(* CODESYS project backup.export

Project tree, tasks and I/O mapping:
  Device : CODESYS Control Win V3 x64, CODESYS, version 3.5.21.10
    application Application
      libraries: Standard, 3.5.18.0 (System)
      task MainTask (cyclic, interval t#20ms, priority 1) calls PLC_PRG
      data type E_Command
      data type E_States
      global variables GVL
      global variables GV_IO
      function BitsToByte [ST]
      function block FB_CircularQueue_Command [ST]: Clear, Dequeue, Enqueue, Peek
      function block FB_ConveyorController [ST]
      function block FB_MachineCenter [ST]: bBusy, bDoorOpened, bEnable, bError, bProduceLids, Progress
      function block FB_OperatorPanel [?]
      function block FB_Positioner [ST]: Clamp, Lift, Lower, Release
      function block FB_PusherController [ST]: Execute
      function block FB_RunTimeTracker [ST]
      function block FB_TwoAxisPaP [ST]: IsMoving, MoveXNeg, MoveXPos, PickUp, ProcessCommand, PutDown
      function block FB_VisionSensorAD [ST]
      program PLC_PRG [ST]
      function block Stage1_PartDetection [ST]: ProcessObjectDetection
      function block Stage2_MC [ST]: ReadyForPart
      function block Stage3_Assembly [ST]
      Symbols
      global variables PersistentVars
    Ethernet : Ethernet, CODESYS, version 4.2.0.0
        settings: IPAddress = [127,0,0,1]; SubnetMask = [255,255,255,0]; GatewayAddress = [0,0,0,0]; MACAddress = [16#00,16#00,16#00,16#00,16#00,16#00]; SaveCommunicationSettings = FALSE; IPAddress = [192,168,0,2]; SubnetMask = [255,255,255,0]; GatewayAddress = [0,0,0,0]
      ModbusTCP_Server_Device : ModbusTCP Server Device, CODESYS, version 4.4.0.0
          settings: DistinctBitAreas = TRUE; Coils Size = 24; Discrete Inputs Size = 19
          input  Application.GV_IO.iMC_Progress : WORD  // Holding Registers.Holding Registers
          input  Application.GV_IO.iBaseVisionSensorBit0 : BOOL  // Coils.Coils.Bit0
          input  Application.GV_IO.iBaseVisionSensorBit1 : BOOL  // Coils.Coils.Bit1
          input  Application.GV_IO.iBaseVisionSensorBit2 : BOOL  // Coils.Coils.Bit2
          input  Application.GV_IO.iBaseVisionSensorBit3 : BOOL  // Coils.Coils.Bit3
          input  Application.GV_IO.iBasePusherBackLimit : BOOL  // Coils.Coils.Bit4
          input  Application.GV_IO.iBasePusherFrontLimit : BOOL  // Coils.Coils.Bit5
          input  Application.GV_IO.iBaseDiffuseSensor : BOOL  // Coils.Coils.Bit6
          input  Application.GV_IO.iEmergencyStopButton : BOOL  // Coils.Coils.Bit7
          input  Application.GV_IO.iResetButton : BOOL  // Coils.Coils.Bit0
          input  Application.GV_IO.iStartButton : BOOL  // Coils.Coils.Bit1
          input  Application.GV_IO.iStopButton : BOOL  // Coils.Coils.Bit2
          input  Application.GV_IO.iMC_Busy : BOOL  // Coils.Coils.Bit3
          input  Application.GV_IO.iMC_Error : BOOL  // Coils.Coils.Bit4
          input  Application.GV_IO.iLidAtPositioner : BOOL  // Coils.Coils.Bit5
          input  Application.GV_IO.iMC_Opened : BOOL  // Coils.Coils.Bit6
          input  Application.GV_IO.iBaseAtPositioner : BOOL  // Coils.Coils.Bit7
          input  Application.GV_IO.iContainerAtExit : BOOL  // Coils.Coils.Bit0
          input  Application.GV_IO.iBasePositionerLimit : BOOL  // Coils.Coils.Bit1
          input  Application.GV_IO.iLidPositionerLimit : BOOL  // Coils.Coils.Bit2
          input  Application.GV_IO.iPaPPartDetected : BOOL  // Coils.Coils.Bit3
          input  Application.GV_IO.iPaPMovingX : BOOL  // Coils.Coils.Bit4
          input  Application.GV_IO.iPaPMovingZ : BOOL  // Coils.Coils.Bit5
          input  Application.GV_IO.iBasePositionerClamped : BOOL  // Coils.Coils.Bit6
          input  Application.GV_IO.iLidPositionerClamped : BOOL  // Coils.Coils.Bit7
          output Application.GV_IO.oResetButtonLight : BOOL  // Discrete Inputs.Discrete Inputs.Bit0
          output Application.GV_IO.oBasePusher : BOOL  // Discrete Inputs.Discrete Inputs.Bit1
          output Application.GV_IO.oStageOneConveyor : BOOL  // Discrete Inputs.Discrete Inputs.Bit2
          output Application.GV_IO.oStartButtonLight : BOOL  // Discrete Inputs.Discrete Inputs.Bit3
          output Application.GV_IO.oStopButtonLight : BOOL  // Discrete Inputs.Discrete Inputs.Bit4
          output Application.GV_IO.oProcessOnLight : BOOL  // Discrete Inputs.Discrete Inputs.Bit5
          output Application.GV_IO.oMC_Start : BOOL  // Discrete Inputs.Discrete Inputs.Bit6
          output Application.GV_IO.oMC_Stop : BOOL  // Discrete Inputs.Discrete Inputs.Bit7
          output Application.GV_IO.oMC_Reset : BOOL  // Discrete Inputs.Discrete Inputs.Bit0
          output Application.GV_IO.oMC_ProduceLids : BOOL  // Discrete Inputs.Discrete Inputs.Bit1
          output Application.GV_IO.oBaseConveyor : BOOL  // Discrete Inputs.Discrete Inputs.Bit2
          output Application.GV_IO.oLidConveyor : BOOL  // Discrete Inputs.Discrete Inputs.Bit3
          output Application.GV_IO.oBasePositionerClamp : BOOL  // Discrete Inputs.Discrete Inputs.Bit4
          output Application.GV_IO.oBasePositionerRaise : BOOL  // Discrete Inputs.Discrete Inputs.Bit5
          output Application.GV_IO.oLidPositionerClamp : BOOL  // Discrete Inputs.Discrete Inputs.Bit6
          output Application.GV_IO.oLidPositionerRaise : BOOL  // Discrete Inputs.Discrete Inputs.Bit7
          output Application.GV_IO.oPaPX : BOOL  // Discrete Inputs.Discrete Inputs.Bit0
          output Application.GV_IO.oPaPZ : BOOL  // Discrete Inputs.Discrete Inputs.Bit1
          output Application.GV_IO.oPaPGrab : BOOL  // Discrete Inputs.Discrete Inputs.Bit2
          unmapped channels: Holding Registers, Input Registers, Coils, Discrete Inputs
*)

// Device/Application/E_Command
{attribute 'qualified_only'}
{attribute 'strict'}
TYPE E_Command :
(
	// Assembler
    eNone,
    eMoveXPos,
    eMoveXNeg,
    eMoveZUp,
    eMoveZDown,
    eGrab,
    eRelease, 
	
	// Positioners
	eClamp, 
	eRaise, 
	eLower
);
END_TYPE

// Device/Application/E_States
{attribute 'qualified_only'}
{attribute 'strict'}
TYPE E_States :
(
	Idle, 
	Running, 
	Waiting, 
	Complete
);
END_TYPE

// Device/Application/GVL
{attribute 'qualified_only'}
VAR_GLOBAL
	SystemEnabled : BOOL;
	SystemFault : BOOL;		// Set by Stage 2
	
	// Trackers
	CurrentRunMinutes : UDINT;
	RejectedPartsCounter : UINT;
	FinishedProductsCounter : UINT;
	ProductionRate : REAL; // Parts/minute
	MaintenenceReset : BOOL;
END_VAR

// Device/Application/GV_IO
{attribute 'qualified_only'}
VAR_GLOBAL
	// INPUTS
	// Vision Sensor
	iBaseVisionSensorBit0: BOOL;
	iBaseVisionSensorBit1: BOOL;
	iBaseVisionSensorBit2: BOOL;
	iBaseVisionSensorBit3: BOOL;
	
	// Pusher
	iBasePusherBackLimit: BOOL;
	iBasePusherFrontLimit: BOOL;
	
	// Diffuser Sensors
	iBaseDiffuseSensor: BOOL;
	iLidAtPositioner: BOOL;
	iBaseAtPositioner : BOOL;
	iContainerAtExit: BOOL;
	
	// Positioners
	iLidPositionerLimit : BOOL;
	iBasePositionerLimit : BOOL;
	iLidPositionerClamped : BOOL;
	iBasePositionerClamped : BOOL;
	
	// Pick & Place Station
	iPaPPartDetected : BOOL;
	iPaPMovingX : BOOL;
	iPaPMovingZ : BOOL;
	
	// Operator Buttons
	iEmergencyStopButton: BOOL;
	iResetButton: BOOL;
	iStartButton: BOOL;
	iStopButton: BOOL;
	
	// Machining Center Sensors
	iMC_Busy: BOOL;
	iMC_Opened: BOOL;
	iMC_Error: BOOL;
	iMC_Progress: WORD;
	
	// OUTPUTS
	// Conveyors
	oStageOneConveyor: BOOL;
	oLidConveyor : BOOL;
	oBaseConveyor : BOOL;
	
	// Pusher
	oBasePusher: BOOL;
	
	// Positioners
	oLidPositionerClamp : BOOL;
	oBasePositionerClamp : BOOL;
	oLidPositionerRaise : BOOL;
	oBasePositionerRaise : BOOL;
	
	// Pick & Place
	oPaPX : BOOL;
	oPaPZ : BOOL;
	oPaPGrab : BOOL;
	
	// Operator Panel lights
	oResetButtonLight: BOOL;
	oStartButtonLight: BOOL;
	oStopButtonLight: BOOL;
	oProcessOnLight: BOOL;
	
	// Machining Center
	oMC_Start: BOOL;
	oMC_Stop: BOOL;
	oMC_Reset: BOOL;
	oMC_ProduceLids: BOOL;
END_VAR

// Device/Application/PersistentVars
{attribute 'qualified_only'}
VAR_GLOBAL PERSISTENT RETAIN
	// Generated instance path of persistent variable
	PLC_PRG.ProcessTimer.iPersistentCounterRunTime: UDINT;
END_VAR

// Device/Application/PLC_PRG
PROGRAM PLC_PRG
VAR
	Operator : FB_OperatorPanel;
	ProcessTimer : FB_RunTimeTracker;
	Stage1 : Stage1_PartDetection;
	Stage2 : Stage2_MC;
	Stage3 : Stage3_Assembly;
END_VAR

// Map IO to Function Blocks
// Operator panel
Operator(
	StartButton := GV_IO.iStartButton, 
	StopButton := GV_IO.iStopButton,
	ResetButton := GV_IO.iResetButton,
	Fault := GVL.SystemFault,
	eStopButton := GV_IO.iEmergencyStopButton);

GV_IO.oProcessOnLight := Operator.ProcessOn;
GV_IO.oStopButtonLight := Operator.ProcessOn;
GV_IO.oResetButtonLight := Operator.ResetButtonLight;
GV_IO.oStartButtonLight := Operator.StartButtonLight;

GVL.SystemFault := Operator.SystemFault;
GVL.SystemEnabled := Operator.ProcessOn;

// Process timer
ProcessTimer(iRun := GVL.SystemEnabled);

// Stage 1 - Part Detection and Processing
Stage1(
	iVisionSensorBit0 := GV_IO.iBaseVisionSensorBit0,
	iVisionSensorBit1 := GV_IO.iBaseVisionSensorBit1,
	iVisionSensorBit2 := GV_IO.iBaseVisionSensorBit2,
	iVisionSensorBit3 := GV_IO.iBaseVisionSensorBit3,
	iPusherBackLimit := GV_IO.iBasePusherBackLimit,
	iPusherFrontLimit := GV_IO.iBasePusherFrontLimit,
	iPusherEntrySensor := GV_IO.iBaseDiffuseSensor);
	
GV_IO.oBasePusher := Stage1.oPusher;
GV_IO.oStageOneConveyor := Stage1.oConveyor;

// Stage 2 - Machining Center
Stage2(
	iBusy := GV_IO.iMC_Busy,
	iOpened := GV_IO.iMC_Opened, 
	iError := GV_IO.iMC_Error, 
	iProgress := GV_IO.iMC_Progress);
	
GV_IO.oMC_ProduceLids := Stage2.oProduceLids;
GV_IO.oMC_Reset := Stage2.oReset;
GV_IO.oMC_Start := Stage2.oStart;
GV_IO.oMC_Stop := Stage2.oStop;

// Pass Ready flag to Stage 1
Stage1(iStage2Ready := Stage2.ReadyForPart);

// Stage 3 - Assembly
Stage3(
	iLidAtClampEntry := GV_IO.iLidAtPositioner, 
	iBaseAtClampEntry := GV_IO.iBaseAtPositioner, 
	iExitSensor := GV_IO.iContainerAtExit, 
	iLidClampLimit := GV_IO.iLidPositionerLimit, 
	iBaseClampLimit := GV_IO.iBasePositionerLimit, 
	iLidClamped := GV_IO.iLidPositionerClamped, 
	iBaseClamped := GV_IO.iBasePositionerClamped,
	iAssemPartDetected := GV_IO.iPaPPartDetected, 
	iAssemIsMovingX := GV_IO.iPaPMovingX, 
	iAssemIsMovingZ := GV_IO.iPaPMovingZ);
	
GV_IO.oLidConveyor := Stage3.oLidConveyor;
GV_IO.oBaseConveyor := Stage3.oBaseConveyor;
GV_IO.oLidPositionerClamp := Stage3.oLidClamp;
GV_IO.oBasePositionerClamp := Stage3.oBaseClamp;
GV_IO.oLidPositionerRaise := Stage3.oLidPositionerRaise;
GV_IO.oBasePositionerRaise := Stage3.oBasePositionerRaise;
GV_IO.oPaPX := Stage3.oAssemMoveX;
GV_IO.oPaPZ := Stage3.oAssemMoveZ;
GV_IO.oPaPGrab := Stage3.oAssemGrab;

END_PROGRAM

// Device/Application/FB_OperatorPanel
FUNCTION_BLOCK FB_OperatorPanel
VAR_INPUT
	StartButton : BOOL;
	StopButton : BOOL;
	ResetButton : BOOL;
	Fault : BOOL;
	eStopButton : BOOL := TRUE;
END_VAR
VAR_OUTPUT
	ProcessOn : BOOL;
	SystemFault : BOOL;
	StartButtonLight : BOOL;
	StopButtonLight : BOOL;
	ResetButtonLight : BOOL;
END_VAR
VAR
	EmergencyStop : BOOL;
END_VAR

(* body of a kind this reader does not render *)

END_FUNCTION_BLOCK

// Device/Application/FB_RunTimeTracker
// Tracks time that iRun is on in minutes in a persistent variable
FUNCTION_BLOCK FB_RunTimeTracker
VAR_INPUT
	iRun : BOOL;		// Process On signal
END_VAR
VAR
	RunTimer : TON;
	R_Run : R_TRIG;
	CurrentMinuteCounter : UDINT;
	TotalMinuteCounter : UDINT;
	R_Reset : R_TRIG;
END_VAR
VAR PERSISTENT
	iPersistentCounterRunTime : UDINT;	// Used to track time since last maintenance
END_VAR

// Run timer when the process is on
RunTimer(IN := iRun, PT := T#60S);

// Check for reset signal
R_Reset(CLK := GVL.MaintenenceReset);
IF R_Reset.Q THEN
	iPersistentCounterRunTime := 0;
END_IF

R_Run(CLK := iRun);
IF R_Run.Q THEN
	CurrentMinuteCounter := 0;	// Reset counter
END_IF

IF RunTimer.Q THEN
	iPersistentCounterRunTime := iPersistentCounterRunTime + 1;
	CurrentMinuteCounter := CurrentMinuteCounter + 1;
	RunTimer(IN := FALSE);	// Reset timer
END_IF

GVL.CurrentRunMinutes := CurrentMinuteCounter;

END_FUNCTION_BLOCK

// Device/Application/Stage1_PartDetection
// FB Controller for the First Stage of the production process (item detection, rejection, and conveyor control)
// - Monitor sensor inputs (Vision sensor, actuator limit switches)
// - Control outputs  (conveyor motor, pusher actuator)
// - Reject metal raw materials by pushing them off the conveyor, while accepting blue materials
// - All outputs are disabled if GV_Flags.SystemEnabled is FALSE
// States:
// - IDLE: Enter RUNNING state if start trigger is TRUE and Stage 2 is ready for material
// - RUNNING: Conveyor on, reject metal raw materials, Enter IDLE if Stage 2 not ready for material
FUNCTION_BLOCK Stage1_PartDetection
VAR_INPUT
	iStage2Ready : BOOL;			// Ready signal from Stage 2
	iVisionSensorBit0 : BOOL;		// LSB, Vision Sensor output
	iVisionSensorBit1 : BOOL;
	iVisionSensorBit2 : BOOL;
	iVisionSensorBit3 : BOOL;		// MSB
	iPusherBackLimit : BOOL;		// Back (reset) position actuator limit switch (NO)
	iPusherFrontLimit : BOOL;		// Front (extended) position actuator limit switch (NO)
	iPusherEntrySensor : BOOL;		// True when object is detected at the entrance of the pusher
END_VAR
VAR_OUTPUT
	oConveyor : BOOL;				// Turn on conveyor motor when TRUE
	oPusher : BOOL;					// Extend pusher arm when TRUE
END_VAR

VAR
	SystemOn: BOOL;					// Local system enabled flag
	ConveyorOn : BOOL;				// Conveyor on signal
	E_State : E_States := E_States.Idle;			// Set intial state
	Reject : BOOL;					// Set in 'ProcessObjectDetection'
	R_PusherEntry : R_TRIG;

	// Controllers
	Pusher : FB_PusherController;
	Conveyor : FB_ConveyorController;
	VisionSensor : FB_VisionSensorAD;
END_VAR

// Check if system is enabled
SystemOn := GVL.SystemEnabled;

// Instantiate Controller FBs
Conveyor(iRun := ConveyorOn);
oConveyor := Conveyor.oRun;
Pusher(iFrontLimit := iPusherFrontLimit, iBackLimit := iPusherBackLimit);
oPusher := Pusher.oPush;
VisionSensor(iBit0 := iVisionSensorBit0, iBit1 := iVisionSensorBit1, iBit2 := iVisionSensorBit2, iBit3 := iVisionSensorBit3);

// Rising triggers
R_PusherEntry(CLK := iPusherEntrySensor);

// Safety stop
IF NOT SystemOn THEN
	E_State := E_States.Idle;
END_IF

CASE E_State OF
	E_States.Idle : 
		ConveyorOn := FALSE;
		IF SystemOn AND iStage2Ready THEN
			E_State := E_States.Running;
		END_IF
	E_States.Running :  
		ConveyorOn := TRUE;
		// Process Vision Sensor Output
		THIS^.ProcessObjectDetection();
		
		// If object should be rejected, wait for it to be at the entrance of pusher before executing
		IF Reject AND R_PusherEntry.Q THEN
			GVL.RejectedPartsCounter := GVL.RejectedPartsCounter + 1;	// Increment counter
			Pusher.Execute();
			Reject := FALSE;	// Reset Reject flag
		END_IF
		
		IF NOT SystemOn OR NOT iStage2Ready THEN
			E_State := E_States.Idle;
		END_IF
END_CASE

// Processes sensor output
// When an object is detected, determines whether it should be accepted or rejected
// If part is to be rejected, pushes the part off the conveyor
METHOD ProcessObjectDetection : BOOL
VAR
	Object: STRING;
END_VAR
IF VisionSensor.bObjectDetected THEN
	Object := VisionSensor.sObjectDetected;
	// Check if object should be rejected
	IF Object = 'metal raw material' OR Object = 'unknown' THEN
		Reject := TRUE;
	END_IF
END_IF
END_METHOD

END_FUNCTION_BLOCK

// Device/Application/FB_PusherController
// FB Controller to control the FactoryIO pneumatic arm pusher
// METHOD: Execute() - Initiates a push. Arm fully extends then retraces back to reset position. 
FUNCTION_BLOCK FB_PusherController
VAR_INPUT
	iFrontLimit : BOOL;		// Front (extended) position limit switch (NO)
	iBackLimit : BOOL;		// Back (reset) position limit switch (NO)
END_VAR
VAR_OUTPUT
	oPush : BOOL;			// Extend arm (when TRUE)
END_VAR
VAR
	PushRequest : BOOL;		// Latch to track push operation
END_VAR

IF PushRequest AND GVL.SystemEnabled THEN
	oPush := TRUE;		// Turn push motor on
	
	IF iFrontLimit THEN // Stop pushing if arm is fully extended
		oPush := FALSE;
		PushRequest := FALSE;
	END_IF
ELSE
	oPush := FALSE;		// Turn push motor off
END_IF

METHOD Execute : BOOL
IF NOT PushRequest AND iBackLimit THEN	// Only push if arm is in reset position
	PushRequest := TRUE;
END_IF
END_METHOD

END_FUNCTION_BLOCK

// Device/Application/FB_ConveyorController
// FB controller to operate the FactoryIO conveyors
FUNCTION_BLOCK FB_ConveyorController	
VAR_INPUT
	iRun : BOOL;	// Run the conveyor
END_VAR
VAR_OUTPUT
	oRun : BOOL;	// Turn on the motor
END_VAR
VAR
END_VAR

// Safety stop
IF NOT GVL.SystemEnabled THEN
	oRun := FALSE;
ELSE
	oRun := iRun;
END_IF

END_FUNCTION_BLOCK

// Device/Application/FB_VisionSensorAD
// FB Controller to decode sensor output from the vision sensor in FactoryIO
// Sensor must be configured to 'All Digital' mode to output 4 bit sequences
FUNCTION_BLOCK FB_VisionSensorAD
VAR_INPUT
	iBit0 : BOOL;	// LSB, 4 sensor output bits from vision sensor 
	iBit1 : BOOL;
	iBit2 : BOOL;
	iBit3 : BOOL;	// MSB
END_VAR
VAR_OUTPUT
	bObjectDetected : BOOL;		// TRUE when the sensor detects something
	sObjectDetected : STRING;	// The object being detected
END_VAR
VAR
	ObjectCode : BYTE;			// Reconstructed bitwise code
END_VAR

// Reconstruct the object code
ObjectCode := BitsToByte(Bit0 := iBit0, Bit1 := iBit1, Bit2 := iBit2, Bit3 := iBit3);

// Decode the result
CASE ObjectCode OF
	0 : sObjectDetected := 'none';
	1 : sObjectDetected := 'blue raw material';
	2 : sObjectDetected := 'blue product lid';
	3 : sObjectDetected := 'blue product base';
	4 : sObjectDetected := 'green raw material';
	5 : sObjectDetected:= 'green product lid';
	6 : sObjectDetected := 'green product base';
	7 : sObjectDetected := 'metal raw material';
	8 : sObjectDetected:= 'metal product lid';
	9 : sObjectDetected := 'metal product base';
ELSE
	sObjectDetected := 'unknown';	
END_CASE

IF sObjectDetected = 'none' THEN
	bObjectDetected := FALSE;
ELSE
	bObjectDetected := TRUE;
END_IF

END_FUNCTION_BLOCK

// Device/Application/BitsToByte
// Converts upto 8 bits into a single byte data type
FUNCTION BitsToByte : BYTE
VAR_INPUT
	Bit0: BOOL := 0;	// LSB
	Bit1: BOOL := 0;
	Bit2: BOOL := 0;
	Bit3: BOOL := 0;
	Bit4: BOOL := 0;
	Bit5: BOOL := 0;
	Bit6: BOOL := 0;
	Bit7: BOOL := 0;	// MSB
END_VAR

// Reconstruct byte useing bitwise shifting
BitsToByte := 
    SHL(TO_BYTE(Bit7), 7) OR
    SHL(TO_BYTE(Bit6), 6) OR
    SHL(TO_BYTE(Bit5), 5) OR
    SHL(TO_BYTE(Bit4), 4) OR
    SHL(TO_BYTE(Bit3), 3) OR
    SHL(TO_BYTE(Bit2), 2) OR
    SHL(TO_BYTE(Bit1), 1) OR
    TO_BYTE(Bit0);

END_FUNCTION

// Device/Application/Stage2_MC
// FB Controller for Stage 2 (Machining Center - MC)
// - Machines raw materials into product bases
// - Manage internal state transisitions using a state machine
// - Sets local 'readyForPart' flag to signal upstream to provide raw material
// - All outputs are disabled if GV_Flags.SystemEnabled is FALSE
// - Sets fault flag if raw material doesn't arrive at entrance within time limit, or incorrect material, requires reset by operator
// States:
// - IDLE: Enter WAITING if system is enabled
// - WAITING: Send start signal to the MC, if MC is busy reset 'ReadyForPart' flag and enter RUNNING
// - RUNNING: Enter COMPLETE when MC stops being busy
// - COMPLETE: Set 'ReadyForPart" flag, enter WAITING if system is still on, else IDLE
FUNCTION_BLOCK Stage2_MC
VAR_INPUT	
	iBusy : BOOL;					// Machining Station is currently processing
	iOpened : BOOL;					// CNC door open
	iError : BOOL;					// Non-raw material detected at station entrance
	iProgress : WORD;				// CNC progress (0 - 100)
END_VAR
VAR_OUTPUT
	oStart: BOOL;					// Start signal for MC, starts machining when part is detected at entry
	oStop: BOOL;					// MC Stop signal
	oReset: BOOL;					// MC Reset signal
	oProduceLids: BOOL;				// TRUE: MC produces lids, FALSE: MC produces bases
END_VAR
VAR
	SystemOn : BOOL;						// Local SystemEnable flag
	E_State : E_States := E_States.Idle;	// Initiate to IDLE
	bReadyForPart: BOOL := TRUE; 			// Local flag signals Stage One to provide raw material
	FaultTimer : TON;						// Timer for waiting for parts to arrive
	bTimerOn : BOOL;						// Used to start the fault timer
	
	MC_Controller : FB_MachineCenter;
END_VAR
VAR CONSTANT
	FaultTimeS : TIME := T#20S;
END_VAR

// Check system is enabled
SystemOn := GVL.SystemEnabled;

// Instantiate Machining Center
MC_Controller(
	iBusy := iBusy, 
	iOpened := iOpened, 
	iError := iError, 
	iProgress := iProgress);
	oStart := MC_Controller.oStart;
	oStop := MC_Controller.oStop;
	oReset := MC_Controller.oReset;
	oProduceLids := MC_Controller.oProduceLids;
	
// Set production type (bases)
MC_Controller.bProduceLids := FALSE;

// If material is incorrect or doesn't arrive
FaultTimer(IN := bTimerOn, PT := FaultTimeS);
IF FaultTimer.Q OR iError THEN
	GVL.SystemFault := TRUE;
	FaultTimer(IN := FALSE);	// Reset fault timer
	bTimerOn := FALSE;
END_IF

// Safety stop
IF NOT SystemOn THEN
	E_State := E_States.Idle;
END_IF

CASE E_State OF
	E_States.Idle :
		MC_Controller.bEnable := FALSE;
		IF SystemOn THEN
			E_State := E_States.Waiting;
		END_IF
	E_States.Waiting:				// Wait for MC to start
		MC_Controller.bEnable := TRUE;
		bTimerOn := TRUE;				// Start fault timer
		IF MC_Controller.bBusy THEN
			bTimerOn := FALSE;
			bReadyForPart := FALSE;
			E_State := E_States.Running;
		END_IF
	E_States.Running:
		IF NOT MC_Controller.bBusy THEN
			E_State := E_States.Complete;
		END_IF
	E_States.Complete:
		bReadyForPart := TRUE;
		E_State := E_States.Idle;
END_CASE

PROPERTY ReadyForPart : BOOL
GET
ReadyForPart := bReadyForPart;
END_GET
END_PROPERTY

END_FUNCTION_BLOCK

// Device/Application/FB_MachineCenter
// FB Controller for the FactoryIO Machining Station
// Robotic arm transports raw material to CNC machine when material is detected and oStart is TRUE
// Part detection is handled internally by FactoryIO
// iError is set when a non-material part is detected at entrance
// Proprties used to set/get Enabled, DoorOpened, Error, IsBusy, ProduceLids, and CNC Progress
FUNCTION_BLOCK FB_MachineCenter
VAR_INPUT
	iBusy : BOOL;				// TRUE when the station is processing raw material
	iOpened : BOOL;				// True when CNC machine door is open
	iError : BOOL;				// True when a non-material part is detected at entry
	iProgress : WORD;			// CNC machining progress (0 - 100)
END_VAR
VAR_OUTPUT
	oStart: BOOL;				// Start signal for MC, starts machining when part is detected at entry
	oStop: BOOL;				// MC Stop signal
	oReset: BOOL;				// MC Reset signal
	oProduceLids: BOOL;			// TRUE: MC produces lids, FALSE: MC produces bases
END_VAR
VAR
	bEnabled : BOOL;			// Enable/Disable Machining Station
	bProduction : BOOL;			// TRUE: Lids, FALSE: Bases
	bIsError : BOOL;			// True when a non-material part is detected at entry
	bIsDoorOpened : BOOL;		// True when CNC machine door is open
END_VAR

// Map variables to outputs
oStart := bEnable;
oProduceLids := bProduction;

// Safety stop
IF NOT GVL.SystemEnabled THEN
	oStop := TRUE;
ELSE
	oStop := FALSE;
END_IF

PROPERTY bBusy : BOOL
GET
bBusy := iBusy;
END_GET
END_PROPERTY

PROPERTY bDoorOpened : BOOL
GET
bDoorOpened := iOpened;
END_GET
END_PROPERTY

PROPERTY bEnable : BOOL
GET
bEnable := bEnabled;
END_GET
SET
bEnabled := bEnable;
END_SET
END_PROPERTY

PROPERTY bError : BOOL
GET
bError := iError;
END_GET
END_PROPERTY

PROPERTY bProduceLids : BOOL
GET
bProduceLids := bProduction;
END_GET
SET
bProduction := bProduceLids;
END_SET
END_PROPERTY

PROPERTY Progress : WORD
GET
Progress := iProgress;
END_GET
END_PROPERTY

END_FUNCTION_BLOCK

// Device/Application/Stage3_Assembly
// FB Controller for Stage 3 - Assembly
// - Assembles product lids and bases into containers using Two-Axis Pick and Place Station
// - Waits for product parts to be ready on their respective conveyors
// - Secures parts with Poistioners (Clamp actuator)
// - All outputs are disabled if GV_Flags.SystemEnabled is FALSE
// States:
// - IDLE: Enter WAITING if system is enabled
// - WAITING: Wait for product parts to be at the positioners
// - RUNNING: Clamp the products to secure them, disable conveyor belts, and assemble into a container
// - COMPLETE: Raises Positioner to allow finished product through

FUNCTION_BLOCK Stage3_Assembly
VAR_INPUT
	iLidAtClampEntry : BOOL;			// Lid at positioner
	iBaseAtClampEntry : BOOL;			// Base at positioner
	iExitSensor : BOOL;					// Container at exit
	iLidClampLimit : BOOL;				// Lid positioner verticle limit switch
	iBaseClampLimit : BOOL;				// Base positioner verticle limit switch
	iLidClamped : BOOL;					// Lid Positier is clamped
	iBaseClamped : BOOL;				// Base positioner is clamped
	iAssemPartDetected : BOOL;			// Part detected in assemblers 'hand'
	iAssemIsMovingX : BOOL;				// Assembler moving in the x-direction
	iAssemIsMovingZ : BOOL;				// Assembler moving in the z-direction
END_VAR
VAR_OUTPUT
	oLidConveyor : BOOL;				// Lid conveyor motor control
	oBaseConveyor : BOOL;				// Base conveyor motor control
	oLidClamp : BOOL;					// Lid Positioner clamp control
	oBaseClamp : BOOL;					// Base positioner clamp control
	oLidPositionerRaise : BOOL;			// Lid positioner raise control
	oBasePositionerRaise : BOOL;		// Base positioner raise control
	oAssemMoveX : BOOL;					// Assembler move x-direction control
	oAssemMoveZ : BOOL;					// Assembler move z-direction control
	oAssemGrab : BOOL;
END_VAR
VAR
	// FB Controllers
	LidConveyor : FB_ConveyorController;
	BaseConveyor : FB_ConveyorController;
	LidPositioner : FB_Positioner;
	BasePositioner : FB_Positioner;
	Assembler : FB_TwoAxisPaP;
	
	SystemOn : BOOL;						// Local System enabled flag
	E_State : E_States := E_States.Idle;	// Initiate State to IDLE
	
	// Falling triggers
	F_LidAtEntry : F_TRIG;
	F_BaseAtEntry : F_TRIG;
	F_ExitSensor : F_TRIG;
	
	// Internal flags
	LidReady : BOOL;
	BaseReady : BOOL;
	LidConveyorOn : BOOL;
	BaseConveyorOn : BOOL;
END_VAR

// Check system is enabled
SystemOn := GVL.SystemEnabled; 

// Instantiate Controller FBs
 LidConveyor(iRun := LidConveyorOn);
 BaseConveyor(iRun := BaseConveyorOn);
 oLidConveyor := LidConveyor.oRun;
 oBaseConveyor := BaseConveyor.oRun;
 
 // Positioners
 LidPositioner(VerticleLimit := iLidClampLimit, iClamped := iLidClamped);
 BasePositioner(VerticleLimit := iBaseClampLimit, iClamped := iBaseClamped);
 
 oLidClamp := LidPositioner.oClamp;
 oLidPositionerRaise := LidPositioner.oRaise;
 oBaseClamp := BasePositioner.oClamp;
 oBasePositionerRaise := BasePositioner.oRaise;
 
 // Assembler (Two-Axis Pick and Place)
 Assembler(
	iPartDetected := iAssemPartDetected, 
	iMovingX := iAssemIsMovingX, 
	iMovingZ := iAssemIsMovingZ);
	
 oAssemGrab := Assembler.oGrab;
 oAssemMoveX := Assembler.oX;
 oAssemMoveZ := Assembler.oZ;
 
 // Falling edge triggers
 F_LidAtEntry(CLK := iLidAtClampEntry);
 F_BaseAtEntry(CLK := iBaseAtClampEntry);
 F_ExitSensor(CLK := iExitSensor);
 
 CASE E_State OF
	 E_States.Idle:
	 LidConveyorOn := FALSE;
	 BaseConveyorOn := FALSE;
	 	IF SystemOn THEN
			E_State := E_States.Waiting;
		END_IF
	E_States.Waiting:
		// Wait for both product parts to be at positioners
		IF NOT LidReady THEN LidConveyorOn := TRUE; END_IF;
		IF NOT BaseReady THEN BaseConveyorOn := TRUE; END_IF;
	
		// If lid at positioner
		IF F_LidAtEntry.Q THEN
			LidPositioner.Clamp();			// Secure part
			LidConveyorOn := FALSE;			// Stop the conveyor
			LidReady := TRUE; 
		END_IF
		IF F_BaseAtEntry.Q THEN
			BasePositioner.Clamp();			// Secure part
			BaseConveyorOn := FALSE;		// Stop the conveyor
			BaseReady := TRUE; 
		END_IF
		
		// If both parts are ready, begin assembly and transitition to RUNNING state
		IF BaseReady AND LidReady AND SystemOn THEN
			Assembler.MoveXPos();			// Move to lid conveyor
			LidPositioner.Release();		// Release the lid
			Assembler.PickUp();				// Pick up the lid
			Assembler.MoveXNeg();			// Move to base conveyor
			Assembler.PutDown();			// Pace lid on base
			E_State := E_States.Running; 
		END_IF
	E_States.Running: 
		// Wait for assembler to finish
		IF NOT Assembler.bBusy and SystemOn THEN
			BasePositioner.Release();		// Release finished product
			BasePositioner.Lift();			// Allow product through
			BaseConveyorOn := TRUE;			// Turn base conveyor back on
			E_State := E_States.Complete;
		END_IF 
	E_States.Complete: 
		// Reset station once finished product has exited
		IF F_ExitSensor.Q THEN
			GVL.FinishedProductsCounter := GVL.FinishedProductsCounter + 1;	// Increment counter
			// Calculate Production Rate
			IF GVL.CurrentRunMinutes <> 0 THEN
				GVL.ProductionRate := TO_REAL(GVL.FinishedProductsCounter) / TO_REAL(GVL.CurrentRunMinutes);
			END_IF
			BasePositioner.Lower();
			LidReady := FALSE;
			BaseReady := FALSE;
			E_State := E_States.Idle;
		END_IF
 END_CASE

END_FUNCTION_BLOCK

// Device/Application/FB_Positioner
// Controller for FactorIOs Clamp Positioner
FUNCTION_BLOCK FB_Positioner
VAR_INPUT
	VerticleLimit : BOOL;	// True when positioner is at reset or fully extended position
	iClamped : BOOL;		// True when clamping
END_VAR
VAR_OUTPUT
	oClamp : BOOL;			// TRUE: activate clamp
	oRaise : BOOL;			// TRUE: Raises the positioner off the conveyor
	bBusy : BOOL;
END_VAR
VAR	
	SystemOn : BOOL;		// Local SystemEnable flag
	E_State : E_States := E_States.Idle;	// Initiate state to Idle
	
	CommandQueue : FB_CircularQueue_Command;
	CurrentCommand : E_Command;
END_VAR

// Check system is enabled
SystemOn := GVL.SystemEnabled;

// Inlcude IF NOT iClamped when adding safety interlocks
CASE E_State OF
	E_States.Idle:
		IF SystemOn AND NOT CommandQueue.bEmpty THEN
			CurrentCommand := CommandQueue.Dequeue();
			bBusy := TRUE;
			E_State := E_States.Waiting;
			CASE CurrentCommand OF
				E_Command.eClamp: oClamp := TRUE;
				E_Command.eRelease: oClamp :=FALSE;
				E_Command.eRaise: oRaise := TRUE;
				E_Command.eLower: oRaise := FALSE;
			END_CASE
		else
			bBusy := false;
		END_IF
	E_States.Waiting:
		IF NOT VerticleLimit OR CurrentCommand = E_Command.eClamp OR CurrentCommand = E_Command.eRelease THEN
			E_State := E_States.Running;
		END_IF
	E_States.Running:
		IF (CurrentCommand = E_Command.eClamp AND iClamped) OR (CurrentCommand = E_Command.eRelease AND NOT iClamped) THEN
			E_State := E_States.Complete;
		ELSIF CurrentCommand = E_Command.eRaise OR CurrentCommand = E_Command.eLower THEN
			IF VerticleLimit THEN
				E_State := E_States.Complete;
			END_IF
		END_IF
	E_States.Complete:
		CurrentCommand := E_Command.eNone;
		E_State := E_States.Idle;
END_CASE

// Activates the Positioners clamp
METHOD Clamp : BOOL
CommandQueue.Enqueue(E_Command.eClamp);
END_METHOD

// Lifts the positioner
// Allows for a part on a conveyor to pass through
METHOD Lift : BOOL
CommandQueue.Enqueue(E_Command.eRaise);
END_METHOD

// Lowers the positioner to the starting position
METHOD Lower : BOOL
CommandQueue.Enqueue(E_Command.eLower);
END_METHOD

// Deactivates the positioners clamp
METHOD Release : BOOL
CommandQueue.Enqueue(E_Command.eRelease);
END_METHOD

END_FUNCTION_BLOCK

// Device/Application/FB_CircularQueue_Command
// Requires E_Command Enum DUT
FUNCTION_BLOCK FB_CircularQueue_Command
VAR_OUTPUT
    bFull  : BOOL;
    bEmpty : BOOL := TRUE;	// Initialize to True
    iCount : INT;
END_VAR

VAR
	MaxSize : INT := 10; 					// Max size of queue (default 10)
    aQueue : ARRAY[0..10] OF E_Command;		// Size must match MaxSize
    iHead  : INT := 0; 						// Points to first valid element
    iTail  : INT := 0; 						// Points to next free spot
END_VAR

// Clears the queue
// Resets iHead and iTail, bFull and iCount
METHOD Clear : BOOL
iHead := 0;
iTail := 0;
bFull := FALSE;
bEmpty := TRUE;
iCount := 0;
END_METHOD

// Dequeue an item from the queue
// Returns the item
METHOD Dequeue : E_Command
VAR
	cmd : E_Command;
END_VAR
IF iTail = iHead THEN
    // Queue is empty
    Dequeue := E_Command.eNone;
ELSE
    Dequeue := aQueue[iHead];
    iHead := (iHead + 1) MOD MaxSize;
END_IF

bFull := ((iTail + 1) MOD MaxSize = iHead);
iCount := (iTail - iHead + MaxSize) MOD MaxSize;
bEmpty := (iTail = iHead);
END_METHOD

// Adds a command to the queue
METHOD Enqueue : BOOL
VAR_INPUT
    cmd : E_Command;
END_VAR
VAR
    nextTail : INT;
END_VAR
nextTail := (iTail + 1) MOD MaxSize;

IF nextTail = iHead THEN
    // Queue is full
    Enqueue := FALSE;
ELSE
    aQueue[iTail] := cmd;
    iTail := nextTail;
    Enqueue := TRUE;
END_IF

bFull := ((iTail + 1) MOD MaxSize = iHead);
bEmpty := (iTail = iHead);
iCount := (iTail - iHead + MaxSize) MOD MaxSize;
END_METHOD

// Returns the first item of the queue without removing it
METHOD Peek : E_Command
IF iTail = iHead THEN
    Peek := E_Command.eNone;
ELSE
    Peek := aQueue[iHead];
END_IF
END_METHOD

END_FUNCTION_BLOCK

// Device/Application/FB_TwoAxisPaP
// Controller for FactoryIOs Two-Axis Pick and Place Station (Digital Configuration)
// - Two positions for each direction; 0: Reset (Starting) position, 1: Extended Position
FUNCTION_BLOCK FB_TwoAxisPaP
VAR_INPUT
	iPartDetected : BOOL;		// True when part is at the gripper
	iMovingX : BOOL;			// Is moving in the X direction
	iMovingZ : BOOL;			// Is moving in teh Z direction
END_VAR
VAR_OUTPUT
	oX : BOOL;					// Extend in the X direction
	oZ : BOOL;					// Extend in the Z direction
	oGrab : BOOL;				// Inititate grab
	bBusy : BOOL;
END_VAR
VAR
	currentCommand : E_Command;
	CommandQueue : FB_CircularQueue_Command;
    state : INT := 0;
END_VAR

CASE state OF
    0: // Idle
        IF GVL.SystemEnabled AND NOT CommandQueue.bEmpty THEN
            currentCommand := CommandQueue.Dequeue();
            state := 1;
            bBusy := TRUE;
			
			ProcessCommand(currentCommand);
		ELSE
			bBusy := FALSE;
        END_IF

    1: // Waiting for motion to start (no movement for grab commands)
        IF IsMoving(currentCommand) OR currentCommand = E_Command.eGrab OR currentCommand = E_Command.eRelease THEN
            state := 2;
        END_IF

    2: // Wait for motion to finish
        IF NOT IsMoving(currentCommand) OR currentCommand = E_Command.eGrab OR currentCommand = E_Command.eRelease THEN
            state := 0;
            currentCommand := E_Command.eNone;
        END_IF
END_CASE

// Returns TRUE if Assmebler is moving based on the command given
METHOD IsMoving : BOOL
VAR_INPUT
	cmd : E_Command;
END_VAR
IF iMovingX OR iMovingZ THEN
	IsMoving := TRUE;
else
	IsMoving := FALSE;
END_IF
END_METHOD

// Moves the assmebler arm to the reset position (x-direction)
METHOD MoveXNeg : BOOL
CommandQueue.Enqueue(E_Command.eMoveXNeg);
END_METHOD

// Moves the assmebler arm to the extended position (x-direction)
METHOD MoveXPos : BOOL
CommandQueue.Enqueue(E_Command.eMoveXPos);
END_METHOD

METHOD PickUp : BOOL
CommandQueue.Enqueue(E_Command.eMoveZDown);
CommandQueue.Enqueue(E_Command.eGrab);
CommandQueue.Enqueue(E_Command.eMoveZUp);
END_METHOD

METHOD ProcessCommand : BOOL
VAR_INPUT
	cmd : E_Command;
END_VAR
// Turn on the relevent output motors
CASE cmd OF
	E_Command.eMoveXPos: oX := TRUE;
	E_Command.eMoveXNeg: oX := FALSE;

	E_Command.eMoveZDown: oZ := TRUE;
	E_Command.eMoveZUp: oZ := FALSE;

	E_Command.eGrab: oGrab := TRUE;
	E_Command.eRelease: oGrab := FALSE;

	E_Command.eNone: // Do nothing
END_CASE
END_METHOD

METHOD PutDown : BOOL
VAR_INPUT
END_VAR
CommandQueue.Enqueue(E_Command.eMoveZDown);
CommandQueue.Enqueue(E_Command.eRelease);
CommandQueue.Enqueue(E_Command.eMoveZUp);
END_METHOD

END_FUNCTION_BLOCK
